(* CoDeSys 2.3.9.50 project: dacha-BC9000.pr6 *)
(* Libraries: PlcHelperBC.lb6 7.5.01 11:03:00, COMlibV2.lb6 25.2.14 08:37:08, ModbusRTU.lb6 13.5.15 12:37:26, standard.lb6 5.6.98 11:03:02 *)

(* Global variable list: Globale_Variablen *)
VAR_GLOBAL

	Clear						: ClearComBuffer;
	TxBufferCom1				: ComBuffer;
	RxBufferCom1				: ComBuffer;
	SerialLineControlCom1			: SerialLineControl;
	ReceiveDataCom1			: ReceiveData;
	SendDataCom1				: SendData;

	Merc_address				: BYTE:=97;

	Modbus						: Modbus_Struct;

	HW_temp_first_floor					AT %IW40:INT;	(* Датчик температуры 1 этаж *)
	HW_temp_second_floor				AT %IW42:INT;	(* Датчик температуры 2 этаж *)
	HW_temp_underfloor					AT %IW44:INT;	(* Датчик температуры подпол 1 этаж *)
	HW_temp_sport						AT %IW46:INT;	(* Датчик температуры спортзал *)

	HW_temp_sport_underfloor				AT %IW48:INT;	(* Датчик температуры подпол спортзал *)
	HW_temp_sauna						AT %IW50:INT;	(* Датчик температуры сауна*)
	HW_temp_street						AT %IW52:INT;	(* Датчик температуры улица *)
	HW_temp_vent						AT %IW54:INT;	(* Датчик температуры притока вентиляции *)

	HW_temp_balkon						AT %IW60:INT;	(* Датчик температуры  *)
	HW_temp_drovnik						AT %IW62:INT;	(* Датчик температуры *)
	HW_temp_sklad						AT %IW64:INT;	(* Датчик температуры  *)
	HW_temp_rezerv						AT %IW66:INT;	(* Датчик температуры  *)


	HW_PIR_terrasa						AT %IX56.0:BOOL;		(*PIR датчик терраса *)
	HW_PIR_zapad						AT %IX56.1:BOOL;		(*PIR датчик запад *)
	HW_PIR_vostok						AT %IX56.2:BOOL;		(*PIR датчик восток *)
	HW_PIR_sport						AT %IX56.3:BOOL;		(*PIR датчик спортзал *)

	HW_GERKON_drovnik					AT %IX56.4:BOOL;		(*Геркон дровник *)
	HW_GERKON_door					AT %IX56.5:BOOL;		(*Геркон дверь *)
	HW_sensor_smoke_1floor				AT %IX56.6:BOOL;		(*Датчик дыма 1 этаж *)
	HW_sensor_smoke_2_3floor			AT %IX56.7:BOOL;		(*Датчик дыма 2 этаж *)

	HW_button_light_garden				AT %IX57.0:BOOL;		(* Кнопка прожектор терраса  *)
	HW_sensor_smoke_sport				AT %IX57.1:BOOL;		(* Кнопка охрана  *)
	HW_button_vorota						AT %IX57.2:BOOL;		(* Кнопка открытия ворот  *)
	HW_button_kalitka					AT %IX57.3:BOOL;		(* Кнопка открытия калитки  *)

	HW_button_poliv_terrasa				AT %IX57.4:BOOL;		(* Кнопка полив терраса 2 часа  *)
	HW_button_poliv_zapad				AT %IX57.5:BOOL;		(* Кнопка полив запад  2 часа  *)
	HW_button_poliv_south				AT %IX57.6:BOOL;		(*  Кнопка полив юг  2 часа  *)
	HW_button_poliv_north					AT %IX57.7:BOOL;		(*  Кнопка полив север  2 часа  *)


	HW_sensor_supply					AT %IX58.0:BOOL;		(* Датчик напряжение  *)
	HW_GERKON_sklad					AT %IX58.1:BOOL;		(*Геркон *)
	HW_PIR_north_zapad					AT %IX58.2:BOOL;		(*PIR датчик  *)
	HW_PIR_north_vostok					AT %IX58.3:BOOL;		(*PIR датчик  *)


	HW_heat_first_floor					AT %QX0.0:BOOL;		(* Отопление 1 этаж *)
	HW_heat_second_floor				AT %QX0.1:BOOL;		(* Отопление 2 этаж *)
	HW_heat_sport						AT %QX0.2:BOOL;		(* Отопление спортзал *)
	HW_heat_underfloor					AT %QX0.3:BOOL;		(* Отопление подпол *)
	HW_heat_sauna						AT %QX0.4:BOOL;		(* Отопление сауна *)
	HW_heat_bathroom					AT %QX0.5:BOOL;		(* Отопление душевая *)
	HW_heat_pipe						AT %QX0.6:BOOL;		(* Отопление водопровод *)
	HW_vent_underfloor					AT %QX0.7:BOOL;		(* Вентиляция подпола *)

	HW_vorota							AT %QX1.0:BOOL;		(* Ворота *)
	HW_kalitka							AT %QX1.1:BOOL;		(* Калитка *)
	HW_pomp_house						AT %QX1.2:BOOL;		(* Насос водоснабжения дома *)
	HW_pomp_garden					AT %QX1.3:BOOL;		(* Насос полива *)
	HW_light_garden						AT %QX1.4:BOOL;		(* Прожектор двор *)
	HW_light_terrasa						AT %QX1.5:BOOL;		(* Свет терраса *)
	HW_light_rezerv						AT %QX1.6:BOOL;		(* Резервное освещение *)
	HW_switch_RS485					AT %QX1.7:BOOL:=TRUE;		(* RS485 line *)


	HW_vent_valve_input					AT %QX2.0:BOOL;		(* Клапан приточной вентиляции *)
	HW_vent_valve_output					AT %QX2.1:BOOL;		(* Клапан вытяжной вентиляции *)
	HW_trans_power						AT %QX2.2:BOOL;		(*Подача тока на трансформатор и реле ТЭН-а *)
	HW_vent_in_heat						AT %QX2.3:BOOL;		(* Подогрев притока - ТЭН *)
	HW_vent_in_heat_level				AT %QX2.4:BOOL;		(* Подогрев притока ночной режим   -5 К ТЭН *)
	HW_vent_in_trans_105_130				AT %QX2.5:BOOL:=FALSE;  (* Напряжение 110 или 130 В *)
	HW_vent_in_trans_160_220				AT %QX2.6:BOOL:=FALSE;  (* Напряжение 160 или 220 В *)
	HW_vent_in_trans_LO_HI				AT %QX2.7:BOOL:=FALSE;  (* Напряжение 110/130  или 160/220 В *)

	HW_poliv_terrasa						AT %QX3.0:BOOL;		(* полив терраса  *)
	HW_poliv_zapad						AT %QX3.1:BOOL;		(* полив запад   *)
	HW_poliv_south						AT %QX3.2:BOOL;		(* полив юг   *)
	HW_poliv_north						AT %QX3.3:BOOL;		(* полив север   *)





END_VAR

(* Global variable list: Variable_Configuration *)
VAR_CONFIG
	RS485read.MB.InData AT %IB32 : MB_KL6inData22B;
	RS485read.MB.OutData AT %QB32 : MB_KL6outData22B;
END_VAR

(* Data type *)
TYPE Modbus_struct :
STRUCT

	(* MEED TO SAVE IN MEMORY*)

	Pomp_house					AT %MB0	:	BOOL;	(*56385*)
	Pomp_garden				AT %MB2	:	BOOL;	(*56386*)
	Light_garden					AT %MB4	:	BOOL;	(*56387*)

	Poliv_zapad					AT %MB6	:	BOOL;	(*56388*)
	Poliv_terrasa					AT %MB8	:	BOOL;	(*56389*)
	Poliv_south					AT %MB10	:	BOOL;	(*56390*)
	Poliv_north					AT %MB12	:	BOOL;	(*56391*)
	Poliv_zapad_minutes			AT %MB14	:	INT;		(*56392*)
	Poliv_terrasa_minutes			AT %MB16	:	INT;		(*56393*)
	Poliv_south_minutes			AT %MB18	:	INT;		(*56394*)
	Poliv_north_minutes			AT %MB20	:	INT;		(*56395*)

	Vent							AT %MB22	:	BOOL;	(*56396*)
	Vent_heat					AT %MB24	:	INT;		(*56397*)
	Vent_heat_level				AT %MB26	:	BOOL;	(*56398*)
	Target_CO2					AT %MB28	:	INT;		(*56399*)

	First_floor_temp_target			AT %MB30	:	INT;		(*56400*)
	Second_floor_temp_target		AT %MB32	:	INT;		(*56401*)
	Sauna_temp_target			AT %MB34	:	INT;		(*56402*)
	Sport_temp_target				AT %MB36	:	INT;		(*56403*)
	Underfloor_temp_target		AT %MB38	:	INT;		(*56404*)
	Underfloor_humidity_target		AT %MB40	:	INT;		(*56405*)

	Security_status				AT %MB42	:	BOOL;		(*56406*)
	Light_reserv					AT %MB44	:	BOOL;		(*56407*)

	(* NOT NEED TO SAVE in MEMORY *)

	First_floor_temp 				AT %MW66	:	REAL;		(*56418*)
	First_floor_hum 				AT %MW70	:	REAL;		(*56420*)
	First_floor_CO2				AT %MW74	:	REAL;		(*56422*)

	Second_floor_temp 			AT %MW78	:	REAL;		(*56424*)
	Second_floor_hum 			AT %MW82	:	REAL;		(*56426*)
	Second_floor_CO2 			AT %MW86	:	REAL;		(*56428*)

	Sport_temp	 				AT %MW90	:	REAL;		(*56430*)
	Sauna_temp	 				AT %MW94	:	REAL;		(*56432*)
	Sklad_temp 					AT %MW98	:	REAL;		(*56434*)
	Sklad_hum 					AT %MW102	:	REAL;		(*56436*)

	Underfloor_temp				AT %MW106	:	REAL;		(*56438*)
	Underfloor_hum				AT %MW110	:	REAL;		(*56440*)

	Sport_underfloor_temp			AT %MW114	:	REAL;		(*56442*)
	Sport_underfloor_hum			AT %MW118	:	REAL;		(*56444*)

	Street_temp					AT %MW122	:	REAL;		(*56446*)
	Street_hum 					AT %MW126	:	REAL;		(*56448*)

	Vent_temp					AT %MW130	:	REAL;		(*56450		*)
	Vent_input_level				AT %MB134	:	INT;			(*56452*)

	Uv1							AT %MW136	:	REAL;		(*56453*)
	Uv2							AT %MW140	:	REAL;		(*56455*)
	Uv3							AT %MW144	:	REAL;		(*56457*)
	Ia1							AT %MW148	:	REAL;		(*56459*)
	Ia2							AT %MW152	:	REAL;		(*56461*)
	Ia3							AT %MW156	:	REAL;		(*56463*)
	Pw_total						AT %MW160	:	REAL;		(*56465*)
	Pw1							AT %MW164	:	REAL;		(*56467*)
	Pw2							AT %MW168	:	REAL;		(*56469*)
	Pw3							AT %MW172	:	REAL;		(*56461*)
	E_T1						AT %MW176	:	REAL;		(*56473*)
	E_T2						AT %MW180	:	REAL;		(*56475		*)

	Poliv_zapad_minutes_est		AT %MB184	:	INT;			(*56477*)
	Poliv_terrasa_minutes_est		AT %MB186	:	INT;			(*56478*)
	Poliv_south_minutes_est		AT %MB188	:	INT;			(*56479*)
	Poliv_north_minutes_est		AT %MB190	:	INT;			(*56480*)

	PIR_terrasa					AT %MB192	:	BOOL;			(*56481*)
	PIR_zapad					AT %MB194	:	BOOL;			(*56482*)
	PIR_vostok					AT %MB196	:	BOOL;			(*56483*)
	PIR_sport					AT %MB198	:	BOOL;			(*56484*)
	PIR_north_zapad				AT %MB200	:	BOOL;			(*56485*)
	PIR_north_vostok				AT %MB202	:	BOOL;			(*56486*)

	GERKON_drovnik				AT %MB204	:	BOOL;			(*56487*)
	GERKON_sklad				AT %MB206	:	BOOL;			(*56488*)
	GERKON_door				AT %MB208	:	BOOL;			(*56489*)
	Smoke_1floor					AT %MB210	:	BOOL;			(*56490*)
	Smoke_2_3floor				AT %MB212	:	BOOL;			(*56491*)
	Smoke_sport					AT %MB214	:	BOOL;			(*56492		= 56385+214/2*)

END_STRUCT
END_TYPE

(* POU MAIN, ST *)
PROGRAM MAIN
VAR
END_VAR
Security;
RS485read;
Poliv;
Ventcontrol;
VentPower;
Thermocontrol;
Buttons;
Power_act;


HW_pomp_house				:=	Modbus.Pomp_house;
HW_light_garden				:=	Modbus.Light_garden;
HW_vorota					:=	HW_button_vorota;




Modbus.First_floor_temp		:=	INT_TO_REAL(HW_temp_first_floor)/10;
Modbus.Second_floor_temp	:=	INT_TO_REAL(HW_temp_second_floor)/10;
Modbus.Sport_temp			:=	INT_TO_REAL(HW_temp_sport)/10;
Modbus.Sauna_temp			:=	INT_TO_REAL(HW_temp_sauna)/10;
Modbus.Underfloor_temp		:=	INT_TO_REAL(HW_temp_underfloor)/10;
Modbus.Street_temp			:=	INT_TO_REAL(HW_temp_street)/10;
Modbus.Vent_temp			:=	INT_TO_REAL(HW_temp_vent)/10;

Modbus.Pw1					:=	Modbus.Uv1*Modbus.Ia1;
Modbus.Pw2					:=	Modbus.Uv2*Modbus.Ia2;
Modbus.Pw3					:=	Modbus.Uv3*Modbus.Ia3;
Modbus.Pw_total				:=	Modbus.Pw1+Modbus.Pw2+Modbus.Pw3;
END_PROGRAM

(* POU Security, ST *)
PROGRAM Security
VAR
END_VAR
Modbus.PIR_terrasa			 :=HW_PIR_terrasa;
Modbus.PIR_zapad			 :=HW_PIR_zapad;
Modbus.PIR_vostok 			 :=HW_PIR_vostok;
Modbus.PIR_sport				 :=HW_PIR_sport;
Modbus.PIR_north_zapad		 :=HW_PIR_north_zapad;
Modbus.PIR_north_vostok		 :=HW_PIR_north_vostok;

Modbus.GERKON_door		 :=HW_GERKON_door;
Modbus.GERKON_drovnik		 :=HW_GERKON_drovnik;
Modbus.GERKON_sklad		 :=HW_GERKON_sklad;


Modbus.Smoke_1floor			 :=HW_sensor_smoke_1floor;
Modbus.Smoke_2_3floor		 :=HW_sensor_smoke_2_3floor;
Modbus.Smoke_sport			 :=HW_sensor_smoke_sport;
END_PROGRAM

(* POU RS485read, ST *)
PROGRAM RS485read
VAR
	MB: ModbusRtuMaster_KL6x22B;

	MBdata : ARRAY [1..2] OF INT;		(* The size of this array can be adapted to the modbus slaves register area *)

	timeoutvalue: TIME := T#500ms;		(* timeout while waiting for an answer of the modbus slave *)

	get_co2_mh_z19b_1floor		: FB_GET_CO2_MH_Z19B;
	get_co2_mh_z19b_1floor_done	: BOOL;
	tmCheck						:TON;

	password_1				: ARRAY [1..6] OF BYTE:=6(1); (* пароль к меркуриям, по умолчанию 6 единиц*)
	crctest					: WORD;
	arrReceive				: ARRAY[1..22] OF BYTE;
	arrSend					: ARRAY[1..22] OF BYTE;

	get_rundata				: FB_GET_RUNDATA;
	get_rundata_done			: BOOL;
	get_energy_E_T1			: FB_GET_ENERGY;
	get_energy_E_T2			: FB_GET_ENERGY;

	sensors_SHT20_v1_id		: ARRAY[1..4] OF BYTE:=16#06, 16#07, 16#08, 16#09;	(* Sensor SHT20 v1 address*)
	sensors_SHT20_v1_hum	: ARRAY[1..4] OF REAL;
	sensors_SHT20_v2_id		: ARRAY[1..2] OF BYTE:=16#0C, 16#0D;				(* Sensor SHT20 v2  address*)
	sensors_SHT20_v2_hum	: ARRAY[1..2] OF REAL;
	sensors_CO2_id			: ARRAY[1..2] OF BYTE:=16#68, 16#65;           (* Senseair S8 address*)
	sensors_CO2_ppm		: ARRAY[1..2] OF REAL;
	get_energy_E_T1_done	: BOOL;
	get_energy_E_T2_done	: BOOL;

	state: INT;
	busy: BOOL;
	FtrigBusy: F_TRIG;
	LastErrorstate: INT;
	LastModbusError: ST_ModbusErrorDiagnostics;
	CounterError: DINT;
	CounterSuccess: DINT;

	Timer1: TON;
	Timer1Q: BOOL;

	i: INT:=1;

END_VAR
tmcheck();

CASE state OF

0:
		MB.ReadRegs(Execute:= FALSE);
		state := 1;
		Clear(Buffer := RxBufferCom1);

1:

			MB.ReadRegs(
			UnitID:= sensors_SHT20_v1_id[i],
			Quantity:= 2,
			MBAddr:= 0,
			cbLength:= 6,
			pMemoryAddr:= ADR(MBdata),
			Execute:= TRUE,
			Timeout:= timeoutvalue,
			Busy => busy,
		);
		IF NOT busy THEN
			IF (mb.Error = FALSE ) THEN
				sensors_SHT20_v1_hum[i]:=INT_TO_REAL(MBdata[2])/10;
			END_IF
			i:=i+1;
			MB.ReadRegs(Execute:= FALSE);
			IF (i>4 )	THEN
				i:=1;
				Modbus.First_floor_hum		:=	sensors_SHT20_v1_hum[1];
				Modbus.Second_floor_hum		:=	sensors_SHT20_v1_hum[2];
				Modbus.Underfloor_hum		:=	sensors_SHT20_v1_hum[3];
				Modbus.Sport_underfloor_hum	:=	sensors_SHT20_v1_hum[4];
				state :=2;
			ELSE
				state :=1;
			END_IF
		END_IF

2:

		MB.ReadInputRegs(
			UnitID:= sensors_SHT20_v2_id[i],
			Quantity:= 2,	(* WORDs *)
			MBAddr:= 1,
			cbLength:= 6,
			pMemoryAddr:= ADR(MBdata),
			Execute:= TRUE,
			Timeout:= timeoutvalue,
			Busy => busy,
		);
		IF NOT busy THEN
			IF (mb.Error = FALSE ) THEN
				sensors_SHT20_v2_hum[i]:=INT_TO_REAL(MBdata[2])/10;
			END_IF
			i:=i+1;
			MB.ReadRegs(Execute:= FALSE);
			IF (i>2 )	THEN
				i:=1;
				Modbus.Street_hum		:=	sensors_SHT20_v2_hum[1];
				Modbus.Sklad_hum		:=	sensors_SHT20_v2_hum[2];
				state :=3;
			ELSE
				state :=2;
			END_IF
		END_IF


3:	(* Read MHZ19 CO2 from sensor. Only 1 on RS485 BUS!!!  *)

		tmCheck(in:=FALSE);
		tmCheck(in:=TRUE,pt:=t#2s);
		get_co2_mh_z19b_1floor_done := FALSE;
		get_co2_mh_z19b_1floor( co2=>Modbus.First_Floor_CO2, done=>get_co2_mh_z19b_1floor_done);
		IF get_co2_mh_z19b_1floor_done OR tmcheck.Q THEN
			 state:=4;
		END_IF

4:	(* Read Senseair S8 CO2 from sensors.  *)
		MB.ReadInputRegs(
			UnitID:=sensors_CO2_id[i], (* station address *)
			Quantity:= 1,
			MBAddr:= 3,
			cbLength:= 4,
			pMemoryAddr:= ADR(MBdata),
			Execute:= TRUE,
			Timeout:= timeoutvalue,
			Busy => busy	);
		IF NOT busy THEN
			IF (mb.Error = FALSE ) THEN
				sensors_CO2_ppm[i]	:=	INT_TO_REAL(MBdata[1]);
			END_IF
			i:=i+1;
			MB.ReadRegs(Execute:= FALSE);
			IF (i>2 )	THEN
				i:=1;
				Modbus.Second_floor_CO2		:=	sensors_CO2_ppm[1];

				state :=25;
			ELSE
				state :=4;
			END_IF
		END_IF


25: (*открываем канал*)


	Clear(Buffer := RxBufferCom1);
	arrSend[1]:=Merc_address;
	arrSend[2]:=1; (*код доступа*)
	arrSend[3]:=1; (*Уровень доступа*)

	MEMCPY(ADR(arrSend)+3,ADR(password_1),6); (*пароль*)
	crctest:=F_CRC16(ADR(arrSend),9); (*расчет контрольной суммы*)
	MEMCPY(ADR(arrSend)+9,ADR(crctest),SIZEOF(crctest)); (*прибавление контрольной суммы к запросу*)
	SendDataCom1(pSendData:=ADR(arrSend),Length:=11,TXBuffer:=TxBufferCom1,Busy=>,Error=>);
	tmCheck(in:=FALSE); tmCheck(in:=TRUE,pt:=t#2s); 	(*запуск таймера проверки - потеря связи\обрыв кабеля*)
	state:=26;

26: (*ответ*)
	ReceiveDataCom1(pPrefix:=,LenPrefix:=,pSuffix:=,LenSuffix:=,
	pReceiveData:=ADR(arrReceive),SizeReceiveData:=4,
	Timeout:=t#2s,Reset:=,
	RXbuffer:=RxBufferCom1,
	DataReceived=>,busy=>,Error=>,RxTimeout=>,LenReceiveData=>);
	IF ReceiveDataCom1.Error <> 0 THEN
		state:=888;
	END_IF
	IF receiveDataCom1.DataReceived THEN
		state:=27;
	ELSIF tmcheck.Q THEN
		state:=888;
	END_IF
27: (*проверка ответа*)

	IF arrReceive[1] = Merc_address THEN
		state:= 28;
	ELSE
		state:=888;
	END_IF



28:
		tmCheck(in:=FALSE);
		tmCheck(in:=TRUE,pt:=t#2s);
		get_rundata_done := FALSE;
		get_rundata(k_div:=100,  byte1:=16#8, byte2:=16#16, byte3:=16#11,  data1=>Modbus.UV1,data2=>Modbus.UV2,data3=>Modbus.UV3, done=>get_rundata_done);
		IF get_rundata_done OR  tmcheck.Q THEN
			 state:=29;
		END_IF


 (*запрос на чтение энергии T1
--------------------------------------------------------------------------------------------------------------------------------------------------------------------
*)

29:
		tmCheck(in:=FALSE);
		tmCheck(in:=TRUE,pt:=t#2s);
		get_energy_E_T1_done := FALSE;
		get_energy_E_T1(byte1:=5, byte2:=16#0, byte3:=1,  energy=>Modbus.E_T1, done=>get_energy_E_T1_done);
		IF get_energy_E_T1_done OR  tmcheck.Q THEN
			state:=30;
		END_IF
 (*запрос на чтение энергии T2
--------------------------------------------------------------------------------------------------------------------------------------------------------------------
*)

30:
	tmCheck(in:=FALSE);
		tmCheck(in:=TRUE,pt:=t#2s);
		get_energy_E_T2_done := FALSE;
		get_energy_E_T2(byte1:=5, byte2:=16#0, byte3:=2,  energy=>Modbus.E_T2, done=>get_energy_E_T2_done);
		IF get_energy_E_T2_done OR  tmcheck.Q THEN
			state:=31;
		END_IF

 (*запрос на чтение тока  на всех фазах
--------------------------------------------------------------------------------------------------------------------------------------------------------------------
*)

31:
		tmCheck(in:=FALSE);
		tmCheck(in:=TRUE,pt:=t#2s);
		get_rundata_done := FALSE;
		get_rundata(k_div:=1000, byte1:=16#8, byte2:=16#16, byte3:=16#21,  data1=>Modbus.Ia1,data2=>Modbus.Ia2,data3=>Modbus.Ia3, done=>get_rundata_done);
		IF get_rundata_done OR tmcheck.Q THEN
			state:=888;
		END_IF



888:
		Timer1(IN:=NOT Timer1Q , PT:=T#10s , Q=>Timer1Q , ET=> );
		IF timer1.q THEN
			state:=0;
		END_IF

END_CASE

FtrigBusy(CLK:=mb.BUSY );
IF FtrigBusy.Q THEN
	IF mb.Error THEN
		LastModbusError := mb.ErrorDiagnostics;
		LastErrorstate := state;
		CounterError := CounterError + 1;
	ELSE
		CounterSuccess := CounterSuccess + 1;
	END_IF
END_IF


(*
SerialLinecontrolCom1(
	mode:=SerialLinemode_kl6_22b_standard,
	pComIn:=ADR(RS485read.MB.InData),
	pComOut:=ADR(RS485read.MB.OutData),
	SizeComIn:=SIZEOF(RS485read.MB.OutData),
	TxBuffer:=TxBufferCom1,
	RxBuffer:=RxBufferCom1,
	Error=>,
	errorid=>);
*)
END_PROGRAM

(* POU FB_GET_CO2_MH_Z19B, ST *)
FUNCTION_BLOCK FB_GET_CO2_MH_Z19B
VAR_INPUT

END_VAR

VAR_OUTPUT
	co2				: REAL;
	done			: BOOL;
END_VAR

VAR
	SendBuffer		: ARRAY[0..8] OF BYTE :=16#FF,16#01,16#86,16#00,16#00,16#00,16#00,16#00,16#79;
	ReceiveBuffer	: ARRAY[0..13] OF BYTE;
	Clear			: ClearComBuffer;
	state			: INT:= 0;
	tmcheck			: TON;
	w_CO2		:	WORD;
(*
	Sensor_CO2_high	 			: BYTE;	
	Sensor_CO2_low 				: BYTE;
*)

END_VAR
tmcheck();

CASE state OF

0:
	done:=FALSE;
	Clear(Buffer := RxBufferCom1);
	SendDataCom1(pSendData:=ADR(SendBuffer),length:=9,TXbuffer:=TXBufferCom1,Busy=>,Error=>);
	tmCheck(in:=FALSE);
	tmCheck(in:=TRUE,pt:=t#2s);
	state:=1;

1: (*ответ*)

	ReceiveDataCom1(pPrefix:=,LenPrefix:=,pSuffix:=,LenSuffix:=,pReceiveData:=ADR(ReceiveBuffer),SizeReceiveData:=9,TImeOut:=t#1s,Reset:=,RXbuffer:=RxBufferCom1,DataReceived=>,busy=>,RxTimeout=>,LenReceiveData=>);

	IF ReceiveDataCom1.Error <> 0 THEN
		state:=9;
	END_IF

	IF ReceiveDataCom1.DataReceived THEN
		state:=2;
	ELSIF tmcheck.Q THEN
		 state:=9;
	END_IF;



2:(*расшифровка*)
	IF (ReceiveBuffer [0] = 16#FF AND ReceiveBuffer [1] = 16#86 ) THEN
(*		Sensor_CO2_high := ReceiveBuffer [2];
		Sensor_CO2_low := ReceiveBuffer [3];	*)
		MEMCPY(ADR(w_CO2),ADR(ReceiveBuffer[3]),1);
		MEMCPY(ADR(w_CO2)+1,ADR(ReceiveBuffer[2]),1);
		co2 := WORD_TO_REAL(w_CO2);

(*		IF (WORD_TO_REAL(w_CO2)<>0 AND WORD_TO_REAL(w_CO2)<5001) THEN
			co2 := WORD_TO_REAL(w_CO2);
			state:=10;
		ELSE
			state:=9;
		END_IF
*)

	ELSE
		state:=9;
	END_IF

9:
	co2:=0;
	done := TRUE;
	state:=0;
10:
	done := TRUE;
	state:=0;

END_CASE;
END_FUNCTION_BLOCK

(* POU FB_GET_RUNDATA, ST *)
FUNCTION_BLOCK FB_GET_RUNDATA
VAR_INPUT
	k_div			: INT;
	byte1			: BYTE;
	byte2			: BYTE;
	byte3			: BYTE;

END_VAR

VAR_OUTPUT
	data1			: REAL;
	data2			: REAL;
	data3			: REAL;
	done			: BOOL;
END_VAR

VAR

	Clear			: ClearComBuffer;
	crctest			: WORD;
	arrReceive		: ARRAY[1..12] OF BYTE := 0,0,0,0,0,0,0,0,0,0,0,0;
	arrSend			: ARRAY[1..6] OF BYTE:= 0,0,0,0,0,0;
	state			: INT:= 0;
	dw_DATA		: DWORD:=0;
	tmcheck			: TON;
	CRC_calc		: WORD:=0;
	CRC_get			: WORD:=1;

END_VAR
tmcheck();

CASE state OF

0:

	done:=FALSE;
	Clear(Buffer := RxBufferCom1);

	arrSend[1]:=Merc_address;
	arrSend[2]:=byte1;
	arrSend[3]:=byte2;
	arrSend[4]:=byte3;

	crctest:=F_CRC16(ADR(arrSend), 4);
	MEMCPY(ADR(arrSend)+4,ADR(crctest),2);

	SendDataCom1(pSendData:=ADR(arrSend),length:=6,TXbuffer:=TXBufferCom1 );

	tmCheck(in:=FALSE);
	tmCheck(in:=TRUE,pt:=t#2s);
	state:=1;

1: (*ответ*)

	ReceiveDataCom1(pReceiveData:=ADR(arrReceive),SizeReceiveData:=12,TImeOut:=t#2s,Reset:=,RXbuffer:=RxBufferCom1);

	IF ReceiveDataCom1.Error <> 0 THEN
		state:=9;
	END_IF

	IF ReceiveDataCom1.DataReceived THEN
		state:=2;

	ELSIF tmcheck.Q THEN state:=9;
	END_IF;


2:(*расшифровка*)
	(* arrReceive:=EchoDel(CheckUp:=TRUE, SentA:=arrSend, RecA:=arrReceive, Length:=UDINT_TO_INT(SendDataCom1.Length)); *)
	CRC_calc := F_CRC16(ADR(arrReceive), 10);
	MEMCPY(ADR(CRC_get),ADR(arrReceive[11]),1);
	MEMCPY(ADR(CRC_get)+1,ADR(arrReceive[12]),1);


	IF (  arrReceive[1] = Merc_address  AND CRC_calc = CRC_get ) THEN
		MEMCPY(ADR(dw_DATA),ADR(arrReceive[3]),1);
			MEMCPY(ADR(dw_DATA)+1,ADR(arrReceive[4]),1);
			arrReceive[2]:=arrReceive[2] AND 16#3F;
			MEMCPY(ADR(dw_DATA)+2,ADR(arrReceive[2]),1);
		data1:=DWORD_TO_REAL(dw_DATA)/k_div;

		MEMCPY(ADR(dw_DATA),ADR(arrReceive[6]),1);
			MEMCPY(ADR(dw_DATA)+1,ADR(arrReceive[7]),1);
			arrReceive[5]:=arrReceive[5] AND 16#3F;
			MEMCPY(ADR(dw_DATA)+2,ADR(arrReceive[5]),1);
		data2:=DWORD_TO_REAL(dw_DATA)/k_div;

		MEMCPY(ADR(dw_DATA),ADR(arrReceive[9]),1);
			MEMCPY(ADR(dw_DATA)+1,ADR(arrReceive[10]),1);
			arrReceive[8]:=arrReceive[8] AND 16#3F;
			MEMCPY(ADR(dw_DATA)+2,ADR(arrReceive[8]),1);
		data3:=DWORD_TO_REAL(dw_DATA)/k_div;



			state:=10;
		ELSE state:=9;
	END_IF;

9:
	data1:=0;
	data2:=0;
	data3:=0;
	done := TRUE;
	state:=0;

10:
	done := TRUE;
	state:=0;

END_CASE;
END_FUNCTION_BLOCK

(* POU MB_func/F_CRC16, ST *)
FUNCTION F_CRC16 : WORD
VAR_INPUT
	pData: POINTER TO BYTE;		(* указатель на блок данных *)
	Size: WORD;						(* размер блока  данных *)
END_VAR
VAR
	Cnt: BYTE;							(* счетчик битов *)
END_VAR
F_CRC16 := 16#FFFF;
WHILE Size > 0 DO
	F_CRC16 := F_CRC16 XOR pData^;
	FOR Cnt := 0 TO 7 DO
		IF F_CRC16.0 = 0 THEN
			F_CRC16 := SHR(F_CRC16, 1);
		ELSE
			F_CRC16 := SHR(F_CRC16, 1) XOR 16#A001;
		END_IF
	END_FOR;
	pData := pData + 1;
	Size := Size - 1;
END_WHILE
END_FUNCTION

(* POU FB_GET_ENERGY, ST *)
FUNCTION_BLOCK FB_GET_ENERGY
VAR_INPUT
	byte1			: BYTE;
	byte2			: BYTE;
	byte3			: BYTE;
END_VAR

VAR_OUTPUT
	energy			: REAL;
	done			: BOOL;
END_VAR

VAR

	Clear				: ClearComBuffer;
	crctest				: WORD;
	arrReceive			: ARRAY[1..22] OF BYTE := 0,0,0,0,0,0,0,0,0,0,0,0,0,0,0,0,0,0,0,0,0,0;
	arrSend				: ARRAY[1..22] OF BYTE:= 0,0,0,0,0,0,0,0,0,0,0,0,0,0,0,0,0,0,0,0,0,0;
	state				: INT:= 0;
	dw_DATA			: DWORD:=0;
(*	E_active				: REAL:=0;
	E_reactive			: REAL:=0;
*)
	tmcheck				: TON;
	CRC_calc			: WORD:=0;
	CRC_get				: WORD:=1;
END_VAR
tmcheck();

CASE state OF

0:
	done:=FALSE;
	Clear(Buffer := RxBufferCom1);
	arrSend[1]:=Merc_address;
	arrSend[2]:=byte1;
	arrSend[3]:=byte2;
	arrSend[4]:=byte3;

	crctest:=F_CRC16(ADR(arrSend), 4);
	MEMCPY(ADR(arrSend)+4,ADR(crctest),2);

	SendDataCom1(pSendData:=ADR(arrSend),length:=6,TXbuffer:=TXBufferCom1 );

	tmCheck(in:=FALSE);
	tmCheck(in:=TRUE,pt:=t#2s);
	state:=1;

1: (*ответ*)

	ReceiveDataCom1(pReceiveData:=ADR(arrReceive),SizeReceiveData:=19,TImeOut:=t#2s,Reset:=,RXbuffer:=RxBufferCom1);

	IF ReceiveDataCom1.Error <> 0 THEN
		state:=9;
	END_IF

	IF ReceiveDataCom1.DataReceived THEN
		state:=2;
	ELSIF tmcheck.Q THEN state:=9;
	END_IF;


2:(*расшифровка*)
	CRC_calc := F_CRC16(ADR(arrReceive), 17);
	MEMCPY(ADR(CRC_get),ADR(arrReceive[18]),1);
	MEMCPY(ADR(CRC_get)+1,ADR(arrReceive[19]),1);

	IF (  arrReceive[1] = Merc_address  AND CRC_calc = CRC_get ) THEN
			MEMCPY(ADR(dw_DATA),ADR(arrReceive[4]),2);
			MEMCPY(ADR(dw_DATA)+2,ADR(arrReceive[2]),2);
			energy:=DWORD_TO_REAL(dw_DATA)/1000;(*активная мощ*)
(*
			MEMCPY(ADR(dw_DATA),ADR(arrReceive[12]),2);
			MEMCPY(ADR(dw_DATA)+2,ADR(arrReceive[10]),2);
			E_reactive:=DWORD_TO_REAL(dw_DATA)/1000; (*реактивная мощность*)

(*			energy:=E_active;	*)
			state:=10;
		ELSE state:=9;
	END_IF;
9:
	energy:=0;
	done := TRUE;
	state:=0;
10:
	done := TRUE;
	state:=0;

END_CASE;
END_FUNCTION_BLOCK

(* POU Poliv, ST *)
PROGRAM Poliv
VAR
	TRIG_poliv_terrasa	:	R_TRIG;
	TRIG_poliv_zapad	:	R_TRIG;
	TRIG_poliv_south		:	R_TRIG;
	TRIG_poliv_north		:	R_TRIG;

	Period_pomp_garden_delay	: INT:=15;				(* Задержка включения насоса после сигнала на открытие клапана=15 сек. *)

 	 tTimerValue_zapad			: TIME;
	Timer_poliv_zapad			: TON;
	Timer_poliv_zapadQ			:  BOOL;
	 tTimerValue_zapad_est		: TIME;

	tTimerValue_terrasa			: TIME;
	Timer_poliv_terrasa			: TON;
	Timer_poliv_terrasaQ			:  BOOL;
	tTimerValue_terrasa_est		: TIME;

	 tTimerValue_south			: TIME;
	Timer_poliv_south				: TON;
	Timer_poliv_southQ			:  BOOL;
	 tTimerValue_south_est		: TIME;


 	tTimerValue_north				: TIME;
	Timer_poliv_north				: TON;
	Timer_poliv_northQ			:  BOOL;
 	tTimerValue_north_est			: TIME;

	TON_pomp_garden			: TON ;
	pomp_garden_start			: BOOL;

	tTimerValue					: TIME;
END_VAR
tTimerValue := DINT_TO_TIME(Period_pomp_garden_delay*1000);


Timer_poliv_zapad();
Timer_poliv_terrasa();
Timer_poliv_south();
Timer_poliv_north();

TRIG_poliv_terrasa(CLK :=HW_button_poliv_terrasa);
TRIG_poliv_zapad(CLK :=HW_button_poliv_zapad);
TRIG_poliv_south(CLK :=HW_button_poliv_south);
TRIG_poliv_north(CLK :=HW_button_poliv_north);


IF (TRIG_poliv_terrasa.Q) THEN
	IF (Modbus.Poliv_terrasa = TRUE ) THEN
		Modbus.Poliv_terrasa := FALSE;

	ELSE

		Modbus.Poliv_terrasa := TRUE;
		Modbus.Poliv_terrasa_minutes:=120;
	END_IF

END_IF



IF (TRIG_poliv_zapad.Q) THEN
	IF (Modbus.Poliv_zapad = TRUE ) THEN

		Modbus.Poliv_zapad := FALSE;
	ELSE

		Modbus.Poliv_zapad := TRUE;
		Modbus.Poliv_zapad_minutes:=120;
	END_IF

END_IF


IF (TRIG_poliv_south.Q) THEN
	IF (Modbus.Poliv_south = TRUE ) THEN

		Modbus.Poliv_south := FALSE;
	ELSE

		Modbus.Poliv_south_minutes:=120;
		Modbus.Poliv_south := TRUE;
	END_IF

END_IF


IF (TRIG_poliv_north.Q) THEN
	IF (Modbus.Poliv_north = TRUE ) THEN

		Modbus.Poliv_north := FALSE;
	ELSE

		Modbus.Poliv_north_minutes:=120;
		Modbus.Poliv_north := TRUE;
	END_IF

END_IF


Modbus.Poliv_zapad_minutes_est	:= TIME_TO_INT(tTimerValue_zapad_est)/(60*1000);
Modbus.Poliv_terrasa_minutes_est	:=  TIME_TO_INT(tTimerValue_zapad_est)/(60*1000);
Modbus.Poliv_south_minutes_est	:=  TIME_TO_INT(tTimerValue_south_est)/(60*1000);
Modbus.Poliv_north_minutes_est	:=  TIME_TO_INT(tTimerValue_north_est)/(60*1000);



IF (Modbus.Poliv_zapad = TRUE ) THEN
	tTimerValue_zapad := DINT_TO_TIME(Modbus.Poliv_zapad_minutes*60*1000);
	HW_poliv_zapad	:=	TRUE;
	Timer_poliv_zapad(IN:=NOT Timer_poliv_zapadQ , PT:=tTimerValue_zapad , Q=>Timer_poliv_zapadQ , ET=>tTimerValue_zapad_est );

END_IF
IF (Modbus.Poliv_zapad = FALSE ) THEN
	HW_poliv_zapad	:=	FALSE;
	Timer_poliv_zapadQ := FALSE;
	Timer_poliv_zapad(IN:=FALSE , PT:=T#0ms , Q=>Timer_poliv_zapadQ , ET=>tTimerValue_zapad_est );
END_IF
IF Timer_poliv_zapad.q THEN
	Modbus.Poliv_zapad := FALSE;
	HW_poliv_zapad	:=	FALSE;
END_IF




IF (Modbus.Poliv_terrasa = TRUE ) THEN
	tTimerValue_terrasa := DINT_TO_TIME(Modbus.Poliv_terrasa_minutes*60*1000);
	HW_poliv_terrasa	:=	TRUE;
	Timer_poliv_terrasa(IN:=NOT Timer_poliv_terrasaQ , PT:=tTimerValue_terrasa , Q=>Timer_poliv_terrasaQ , ET=>tTimerValue_terrasa_est );
END_IF
IF (Modbus.Poliv_terrasa = FALSE ) THEN
	HW_poliv_terrasa	:=	FALSE;
	Timer_poliv_terrasaQ := FALSE;
	Timer_poliv_terrasa(IN:=FALSE , PT:=T#0ms , Q=>Timer_poliv_terrasaQ , ET=>tTimerValue_terrasa_est );
END_IF
IF Timer_poliv_terrasa.q THEN
	Modbus.Poliv_terrasa := FALSE;
	HW_poliv_zapad	:=	FALSE;
END_IF



IF (Modbus.Poliv_south = TRUE ) THEN
	tTimerValue_south := DINT_TO_TIME(Modbus.Poliv_south_minutes*60*1000);
	HW_poliv_south	:=	TRUE;
	Timer_poliv_south(IN:=NOT Timer_poliv_southQ , PT:=tTimerValue_south , Q=>Timer_poliv_southQ , ET=>tTimerValue_south_est );
END_IF
IF (Modbus.Poliv_south = FALSE ) THEN
	HW_poliv_south	:=	FALSE;
	Timer_poliv_southQ := FALSE;
	Timer_poliv_south(IN:=FALSE , PT:=T#0ms , Q=>Timer_poliv_southQ , ET=>tTimerValue_south_est );
END_IF
IF Timer_poliv_south.q THEN
	Modbus.Poliv_south := FALSE;
	HW_poliv_south	:=	FALSE;
END_IF



IF (Modbus.Poliv_north = TRUE ) THEN
	tTimerValue_north := DINT_TO_TIME(Modbus.Poliv_north_minutes*60*1000);
	HW_poliv_north	:=	TRUE;
	Timer_poliv_north(IN:=NOT Timer_poliv_northQ , PT:=tTimerValue_north , Q=>Timer_poliv_northQ , ET=>tTimerValue_north_est );
END_IF
IF (Modbus.Poliv_north = FALSE ) THEN
	HW_poliv_north	:=	FALSE;
	Timer_poliv_northQ := FALSE;
	Timer_poliv_north(IN:=FALSE , PT:=T#0ms , Q=>Timer_poliv_northQ , ET=>tTimerValue_north_est );
END_IF
IF Timer_poliv_north.q THEN
	Modbus.Poliv_north := FALSE;
	HW_poliv_north	:=	FALSE;
END_IF






IF ((HW_poliv_zapad=TRUE OR HW_poliv_terrasa=TRUE 	OR HW_poliv_south =	TRUE OR HW_poliv_north = TRUE) AND (HW_pomp_Garden=FALSE)  )  THEN
	pomp_garden_start			:=TRUE;
END_IF


TON_pomp_garden(IN := pomp_garden_start, PT:= tTimerValue);
Modbus.Pomp_garden	 	:= TON_pomp_garden.Q;
HW_Pomp_garden		:= TON_pomp_garden.Q;

IF (HW_poliv_zapad=FALSE AND HW_poliv_terrasa=FALSE 	AND HW_poliv_south = FALSE  AND HW_poliv_north = FALSE)   THEN
	pomp_garden_start		:= FALSE;
	Modbus.Pomp_garden	 	:= FALSE;
	HW_Pomp_garden		:= FALSE;
END_IF
END_PROGRAM

(* POU Ventcontrol, ST *)
PROGRAM VentControl
VAR
	Temperature_max_to_heat	: REAL:=17;		(* Максимальная температура наружнего воздуха при которой разрешено включать воздухонагреватель*)
	gisterezis				: REAL:=0.2;	(* Гистерезис  разрешения включения воздухонагревателя, градусы цельсия *)
	vent_valve_opened	 	: BOOL:=FALSE;	(*После перезагрузки ПЛК считаем что приточный клапан закрыт *)
(*	Period_start_delay		: INT:=60; 	(* Время задержки включения вентилятора после сигнала на открытие приточного клапана, сек *)
(*	Period_stop_delay		: INT:=60;		(* Время задержки отключения вентилятора после сигнала на останов вентиляции - для остужения разогретых ТЭНов воздухонагревателя, сек *)

	Timer1					: TON;		(* Таймер задержки включения вентилятора после сигнала на открытие приточного клапана *)
	Timer2					: TON;		(* Таймер задержки отключения вентилятора после сигнала на останов вентиляции - для остужения разогретых ТЭНов воздухонагревателя *)
	Timer1Q					: BOOL;
	Timer2Q					: BOOL;
(*
	tTimerValue1				: TIME;
	tTimerValue2				: TIME;
*)

END_VAR
(*
tTimerValue1 := DINT_TO_TIME(Period_start_delay*1000);
tTimerValue2 := DINT_TO_TIME(Period_stop_delay*1000);
*)

IF (Modbus.Vent=FALSE) THEN
	HW_vent_in_heat := FALSE;
	vent_valve_opened := FALSE;
	HW_vent_valve_input:=FALSE;
	Timer2(IN:=NOT Timer2Q , PT:=t#60s , Q=>Timer2Q , ET=> );
	IF timer2q THEN
		HW_trans_power:=FALSE;
	END_IF


ELSE
	HW_vent_valve_input:=TRUE;
	HW_vent_valve_output:=TRUE;

	IF (vent_valve_opened = FALSE) THEN		(* change this block if valve has output signal of status: OPEN/CLOSED *)
		Timer1(IN:=NOT Timer1Q , PT:=t#60s , Q=>Timer1Q , ET=> );
		IF timer1.q THEN
			vent_valve_opened := TRUE;
		END_IF
	END_IF

	IF (vent_valve_opened=TRUE) THEN
		HW_trans_power:=TRUE;
(*		IF (HW_vent_reay_pressure=TRUE) THEN	*)

			IF (Modbus.Vent_heat=2) THEN
				IF (Modbus.Street_temp < Temperature_max_to_heat-gisterezis) THEN
					HW_vent_in_heat:=TRUE;
					IF (Modbus.Vent_heat_level=TRUE) THEN
						HW_vent_in_heat_level:=TRUE;
					END_IF
				END_IF
				IF (Modbus.Street_temp > Temperature_max_to_heat+gisterezis) THEN
					HW_vent_in_heat:=FALSE;
				END_IF
			ELSE
				IF (Modbus.Vent_heat=1) THEN
					HW_vent_in_heat:=TRUE;
					IF (Modbus.Vent_heat_level=TRUE) THEN
						HW_vent_in_heat_level:=TRUE;
					ELSE
						HW_vent_in_heat_level:=FALSE;
					END_IF
				END_IF
				IF (Modbus.Vent_heat=0) THEN
					HW_vent_in_heat:=FALSE;
				END_IF
			END_IF
(*		END_IF   *)(*vent_relay_pressure*)
	END_IF (*vent_valve_opened*)
END_IF (*Vent*)
END_PROGRAM

(* POU VentPower, ST *)
PROGRAM VentPower
VAR
	Vent_power			: REAL:=30;  (* После перезагрузки ПЛК задаём начальную мощность условных 30%  *)
	CO2_old				: REAL:=410; (* После перезагрузки ПЛК задаём принудительно последнее значение CO2 = 410 (абсолютно свежий воздух) *)
(*	Period_vent_switch	: INT:=180; (* Частота переключения режимов работы вентилятора по показаниям датчиков CO2, секунды*)
	Timer1				: TON;
	Timer1Q				: BOOL;
	count				: INT:=0;
	CO2_max			: REAL;
(*	tTimerValue			: TIME;	*)

END_VAR
(* tTimerValue := DINT_TO_TIME(Period_vent_switch*1000);  *)

IF (Modbus.Vent =TRUE  ) THEN

	Timer1(IN:=NOT Timer1Q , PT:=t#180s , Q=>Timer1Q , ET=> );

	IF timer1.q THEN
	CO2_max:=MAX (Modbus.First_floor_CO2, Modbus.Second_floor_CO2);

	IF (  (CO2_max >=  CO2_old-10 )  AND ( CO2_max >  INT_TO_REAL(Modbus.Target_CO2)*1.05 ) ) THEN
			Vent_power:=Vent_power+5;
		END_IF
		count:=count+1;

		IF (count = 2)	THEN
			IF (  CO2_max <=  INT_TO_REAL(Modbus.Target_CO2)*0.99) THEN
				Vent_power:=Vent_power-1;
			END_IF
		count:=1;
		END_IF

		IF (Vent_power>80) THEN
			Vent_power:=80;
		END_IF
		IF(Vent_power<20) THEN
			Vent_power:=20;
		END_IF

		IF (Vent_Power > 75 AND Modbus.Street_temp > -10  ) THEN

					Modbus.Vent_input_level:=200;	(*200 м. куб в час при подаче напряжения на вентилятор  220V *)
					HW_vent_in_trans_160_220:=FALSE;
					HW_vent_in_trans_LO_HI:=FALSE;

			ELSIF (Vent_Power>50 AND Modbus.Street_temp > -15) THEN
					Modbus.Vent_input_level:=180; (*200 м. куб в час при подаче напряжения на вентилятор 220V *)
					HW_vent_in_trans_160_220:=FALSE;
					HW_vent_in_trans_LO_HI:=FALSE;

			ELSIF (Vent_Power>35  AND Modbus.Street_temp > -20) THEN

					Modbus.Vent_input_level:=150; (* 150 м. куб в час при подаче напряжения на вентилятор160V *)
					HW_vent_in_trans_160_220:=TRUE;
					HW_vent_in_trans_LO_HI:=FALSE;


			ELSIF (Vent_Power>25 ) THEN

					Modbus.Vent_input_level:=110; (* 110 м. куб в час при подаче напряжения на вентилятор 130V *)
					HW_vent_in_trans_105_130:=FALSE;
					HW_vent_in_trans_LO_HI:=TRUE;


			ELSE
				Modbus.Vent_input_level:=80; (* 80 м. куб в час при подаче напряжения на вентилятор 105V *)
				HW_vent_in_trans_105_130:=TRUE;
				HW_vent_in_trans_LO_HI:=TRUE;


			END_IF

			CO2_old:=CO2_max;

		END_IF	(* Timer1 *)

	ELSE	 (* Vent=TRUE*)


		Modbus.Vent_input_level:=0;

END_IF   (* Vent=TRUE*)
END_PROGRAM

(* POU Thermocontrol, ST *)
PROGRAM Thermocontrol
VAR
	gisterezis		: REAL:=0.2; (*Гистерезис термостата, градусы цельсия *)
	Timer1			: TON;
	Timer1Q			: BOOL;
END_VAR
(*  tTimerValue := DINT_TO_TIME(period_sec*1000); *)



Timer1(IN:=NOT Timer1Q , PT:=t#120s , Q=>Timer1Q , ET=> );
IF timer1.q THEN

	IF (Modbus.First_floor_temp > Modbus.First_floor_temp_target+gisterezis ) THEN
		HW_heat_first_floor:=FALSE;
	ELSIF (Modbus.First_floor_temp <  Modbus.First_floor_temp_target-gisterezis)  THEN
		HW_heat_first_floor:=TRUE;
	END_IF

	IF (Modbus.Second_floor_temp > Modbus.Second_floor_temp_target+gisterezis ) THEN
		HW_heat_Second_floor:=FALSE;
	ELSIF (Modbus.Second_floor_temp <  Modbus.Second_floor_temp_target-gisterezis ) THEN
		HW_heat_Second_floor:=TRUE;
	END_IF

	IF (Modbus.Sport_temp > Modbus.Sport_temp_target+gisterezis ) THEN
		HW_heat_sport:=FALSE;
	ELSIF (Modbus.Sport_temp <  Modbus.Sport_temp_target-gisterezis )  THEN
		HW_heat_sport:=TRUE;
	END_IF

	IF (Modbus.Sauna_temp > Modbus.Sauna_temp_target+gisterezis ) THEN
		HW_heat_Sauna:=FALSE;
	ELSIF (Modbus.Sauna_temp <  Modbus.Sauna_temp_target-gisterezis ) THEN
		HW_heat_Sauna:=TRUE;
	END_IF

	IF (Modbus.Underfloor_temp > Modbus.Underfloor_temp_target+gisterezis AND Modbus.Underfloor_hum < Modbus.Underfloor_humidity_target-1 ) THEN
		HW_heat_underfloor:=FALSE;
	ELSIF ((Modbus.Underfloor_temp <  Modbus.Underfloor_temp_target-gisterezis OR Modbus.Underfloor_hum > Modbus.Underfloor_humidity_target+1) ) THEN
		HW_heat_Underfloor:=TRUE;
	END_IF


END_IF
END_PROGRAM

(* POU Buttons, ST *)
PROGRAM Buttons
VAR

	SW_LIGHT_GARDEN			: SM_BUTT;		(* вкл/откл прожектор *)

END_VAR
SW_LIGHT_GARDEN		(IN:=HW_button_light_garden, IN1:=Modbus.Light_garden, 	Q=>Modbus.Light_garden);		(* Конпка *)
END_PROGRAM

(* POU SM_BUTT, ST *)
FUNCTION_BLOCK SM_BUTT            (* ФУНКЦИОНАЛЬНЫЙ БЛОК ДЛЯ ПРОСТОЙ КНОПКИ *)
    VAR_INPUT
       	IN: BOOL;          	(*ВХОД ЗА КОТОРЫМ МЫ СЛЕДИМ *)
	IN1:BOOL;				(*ВЫХОД ЗА КОТОРЫМ ТОЖЕ СЛЕДИМ*)
    END_VAR

    VAR_OUTPUT
	Q : BOOL;        			(*СОСТОЯНИЕ ВЫХОДА*)
    END_VAR
    VAR
  MEM : BOOL;    			(* ВНУТРЕННЯЯ ПЕРЕМЕННАЯ ДЛЯ ХРАНЕНИЯ СОСТОЯНИЯ КНОПКИ *)
    END_VAR
Q:=IN1;

IF IN AND NOT MEM THEN 	(* ПОЙМАЛИ ПЕРЕДНИЙ ФРОНТ - НАЖАЛИ НА КНОПКУ *)
	Q := NOT IN1;    			(* МЕНЯЕМ СОСТОЯНИЕ ВЫХОДА НА ПРОТИВОПОЛОЖНОЕ *)
END_IF

MEM := IN;                       		(* ЗАПОМИНАЕМ ТЕКУЩЕЕ ЗНАЧЕНИЕ КНОПКИ *)
END_FUNCTION_BLOCK

(* POU Power_act, ST *)
PROGRAM Power_act
VAR
END_VAR
IF (Modbus.Security_status = FALSE AND HW_sensor_supply = FALSE  ) THEN
	Modbus.Light_reserv :=TRUE;
END_IF

IF (Modbus.Security_status = TRUE ) THEN
	Modbus.Light_reserv := FALSE;
END_IF
END_PROGRAM
